    // Build the message NOW, so text and values are from the moment of
    // the fault. PRG_Spray.sErrorText is current: MAIN calls PRG_Spray
    // before this program in the same scan.
    sText := 'SPRAY FAULT ';
    sText := CONCAT(sText, INT_TO_STRING(MAIN.nErrorCode));
    sText := CONCAT(sText, ': ');
    sText := CONCAT(sText, PRG_Spray.sErrorText);
    sText := CONCAT(sText, '\nLevel ');           // '\n' = literal chars
    sText := CONCAT(sText, LREAL_TO_FMTSTR(REAL_TO_LREAL(GVL_IO.rSPXLevel), 1, TRUE));
    sText := CONCAT(sText, ' % / SPX ');
    sText := CONCAT(sText, LREAL_TO_FMTSTR(REAL_TO_LREAL(GVL_IO.rSPXPressure), 2, TRUE));
    sText := CONCAT(sText, ' bar');
    IF fbTime.bValid THEN
        sText := CONCAT(sText, '\n');
        sText := CONCAT(sText, SYSTEMTIME_TO_STRING(fbTime.systemTime));
    END_IF

    // JSON wrapper. The '\n' above is backslash+n (two characters) -
    // JSON turns that into a real newline in the Telegram message.
    // Keep sText plain ASCII without quotes/backslashes, or escape them.
    sPending := '{"chat_id":"';
    sPending := CONCAT(sPending, sChatId);
    sPending := CONCAT(sPending, '","text":"');
    sPending := CONCAT(sPending, sText);
    sPending := CONCAT(sPending, '"}');
    // NOTE: a newer fault overwrites an unsent one (one-slot queue).
END_IF

//==================================================================
// Send state machine: hand over -> wait for the response -> idle.
//==================================================================
CASE eStep OF

    IDLE:
        IF sPending <> '' THEN
            sBody    := sPending;
            sPending := '';
            eStep    := SEND;
        END_IF

    SEND:
        // Retry the handover for up to 10 s (client may still be
        // configuring right after boot), then drop the message.
        tonSendTo(IN := TRUE, PT := T#10S);
        fbRequest.sContentType := 'application/json';
        IF fbRequest.SendRequest(sUri         := sUri,
                                 fbClient     := fbClient,
                                 eRequestType := ETcIotHttpRequestType.HTTP_POST,
                                 pContent     := ADR(sBody),
                                 nContentSize := TO_UDINT(LEN(sBody)),
                                 fbHeader     := 0) THEN
            tonSendTo(IN := FALSE);
            eStep := WAIT_RESPONSE;
        ELSIF tonSendTo.Q THEN
            tonSendTo(IN := FALSE);
            nFailCount := nFailCount + 1;     // never block the machine
            eStep := IDLE;
        END_IF

    WAIT_RESPONSE:
        // bBusy TRUE->FALSE = response received (or the request failed).
        IF NOT fbRequest.bBusy THEN
            nLastStatus := fbRequest.nStatusCode;
            IF fbRequest.bError OR (fbRequest.nStatusCode <> 200) THEN
                nFailCount := nFailCount + 1;
            END_IF
            eStep := IDLE;
        END_IF

END_CASE

END_PROGRAM

// ---- POUs/PRG_StatsLogger.TcPOU
PROGRAM PRG_StatsLogger
VAR
    fbTime     : FB_LocalSystemTime := (bEnable := TRUE, dwCycle := 1);
    tsNow         : TIMESTRUCT;

    // ---- sampling ----
    tonSample  : TON;
    bDue       : BOOL;
    bActive    : BOOL;
    bInWindow  : BOOL;
    tPeriod    : TIME;
    ePrevState : E_SeqState := E_SeqState.eIdle;
    bPrevAuto  : BOOL;

    // ---- time-in-state accumulators (for uptime %) ----
    tonSec     : TON;
    nRunSec    : UDINT;   // resets on PLC restart (by design)
    nIdleSec   : UDINT;
    nFaultSec  : UDINT;

    // ---- line queue (writer drains it; survives short disk hiccups) ----
    aQ         : ARRAY [0..15] OF STRING(255);
    nHead      : INT;
    nTail      : INT;
    nCount     : INT;
    nDropped   : UDINT;

    // ---- file writer state machine ----
    eWr        : (WR_IDLE, WR_OPEN, WR_WRITE, WR_CLOSE);
    fbOpen     : FB_FileOpen;
    fbWrite    : FB_FilePuts;
    fbClose    : FB_FileClose;
    hFile      : UINT;
    bBoot      : BOOL;             // TRUE -> sLogDir='' -> boot folder
    sPath      : STRING(255);
    sLastDate  : STRING(15);
    tonRetry   : TON;
    bBackoff   : BOOL;
    nFailCount : UDINT;
    nLastErrId : UDINT;
    sLastPath  : STRING(255);

    // ---- scratch ----
    sTs        : STRING(63);
    sDate      : STRING(15);
    sFile      : STRING(80);
    sLine      : STRING(255);
    sTail      : STRING(2);
END_VAR

fbTime();

//------------------------------------------------------------------
// 1) time-in-state accumulators (1 s resolution)
//------------------------------------------------------------------
tonSec(IN := NOT tonSec.Q, PT := T#1S);
IF tonSec.Q THEN
    IF MAIN.eState = E_SeqState.eFault THEN
        nFaultSec := nFaultSec + 1;
    ELSIF MAIN.eState = E_SeqState.eIdle THEN
        nIdleSec := nIdleSec + 1;
    ELSE
        nRunSec := nRunSec + 1;
    END_IF
END_IF

//------------------------------------------------------------------
// 2) is logging allowed right now?  (master switch + daily window)
//------------------------------------------------------------------
tsNow := fbTime.systemTime;
IF (GVL_Param.nStatsHourFrom = 0) AND (GVL_Param.nStatsHourTo = 0) THEN
    bInWindow := TRUE;                                   // 24 h logging
ELSIF GVL_Param.nStatsHourFrom <= GVL_Param.nStatsHourTo THEN
    bInWindow := (tsNow.wHour >= INT_TO_WORD(GVL_Param.nStatsHourFrom))
             AND (tsNow.wHour <  INT_TO_WORD(GVL_Param.nStatsHourTo));
ELSE                                                     // window over midnight
    bInWindow := (tsNow.wHour >= INT_TO_WORD(GVL_Param.nStatsHourFrom))
              OR (tsNow.wHour <  INT_TO_WORD(GVL_Param.nStatsHourTo));
END_IF

//------------------------------------------------------------------
// 3) adaptive sample trigger (+ immediate sample on any edge)
//------------------------------------------------------------------
bActive := (MAIN.eState <> E_SeqState.eIdle) AND (MAIN.eState <> E_SeqState.eFault);
tPeriod := SEL(bActive, GVL_Param.tStatsIdle, GVL_Param.tStatsRun);
tonSample(IN := NOT tonSample.Q, PT := tPeriod);
bDue := tonSample.Q;
IF (MAIN.eState <> ePrevState) OR (MAIN.bAutoMode <> bPrevAuto) THEN
    bDue := TRUE;                    // sharp edges on the state timeline
END_IF
ePrevState := MAIN.eState;
bPrevAuto  := MAIN.bAutoMode;

//------------------------------------------------------------------
// 4) build + queue one CSV line
//------------------------------------------------------------------
IF bDue AND bInWindow AND GVL_Param.bStatsEnable AND fbTime.bValid THEN

    // ---- timestamp 'YYYY-MM-DD HH:MM:SS.mmm' (fixed format for Alloy) ----
    sTs := TO_STRING(tsNow.wYear);
    sTs := CONCAT(sTs, SEL(tsNow.wMonth  < 10, '-', '-0'));
    sTs := CONCAT(sTs, TO_STRING(tsNow.wMonth));
    sTs := CONCAT(sTs, SEL(tsNow.wDay    < 10, '-', '-0'));
    sTs := CONCAT(sTs, TO_STRING(tsNow.wDay));
    sDate := sTs;                                        // YYYY-MM-DD
    sTs := CONCAT(sTs, SEL(tsNow.wHour   < 10, ' ', ' 0'));
    sTs := CONCAT(sTs, TO_STRING(tsNow.wHour));
    sTs := CONCAT(sTs, SEL(tsNow.wMinute < 10, ':', ':0'));
    sTs := CONCAT(sTs, TO_STRING(tsNow.wMinute));
    sTs := CONCAT(sTs, SEL(tsNow.wSecond < 10, ':', ':0'));
    sTs := CONCAT(sTs, TO_STRING(tsNow.wSecond));
    sTs := CONCAT(sTs, '.');
    IF tsNow.wMilliseconds < 10 THEN
        sTs := CONCAT(sTs, '00');
    ELSIF tsNow.wMilliseconds < 100 THEN
        sTs := CONCAT(sTs, '0');
    END_IF
    sTs := CONCAT(sTs, TO_STRING(tsNow.wMilliseconds));

    // ---- day rollover: new file name + one header line ----
    IF sDate <> sLastDate THEN
        sLastDate := sDate;
        sFile := CONCAT('machine_stats_', sDate);
        sFile := CONCAT(sFile, '.csv');
        IF GVL_Param.sLogDir = '' THEN
            bBoot := TRUE;
            sPath := sFile;                              // TwinCAT boot folder
        ELSE
            bBoot := FALSE;
            sPath := GVL_Param.sLogDir;
            sTail := RIGHT(sPath, 1);
            IF (sTail <> '\') AND (sTail <> '/') THEN
                sPath := CONCAT(sPath, '/');             // '/' works on Windows too
            END_IF
            sPath := CONCAT(sPath, sFile);
        END_IF
        IF nCount < 16 THEN                              // header line
            aQ[nTail] := '# ts,state,state_n,mode,level_pct,spx_bar,air_bar,pump_hz,err,run_s,idle_s,fault_s';
            nTail := (nTail + 1) MOD 16;
            nCount := nCount + 1;
        END_IF
    END_IF

    // ---- the sample itself ----
    sLine := sTs;
    sLine := CONCAT(sLine, ',');
    sLine := CONCAT(sLine, TO_STRING(MAIN.eState));      // 'eIdle' etc.
    sLine := CONCAT(sLine, ',');
    sLine := CONCAT(sLine, INT_TO_STRING(TO_INT(MAIN.eState)));  // 0/10/../100
    sLine := CONCAT(sLine, SEL(MAIN.bAutoMode, ',MAN', ',AUTO'));
    sLine := CONCAT(sLine, ',');
    sLine := CONCAT(sLine, LREAL_TO_FMTSTR(REAL_TO_LREAL(GVL_IO.rSPXLevel), 1, TRUE));
    sLine := CONCAT(sLine, ',');
    sLine := CONCAT(sLine, LREAL_TO_FMTSTR(REAL_TO_LREAL(GVL_IO.rSPXPressure), 2, TRUE));
    sLine := CONCAT(sLine, ',');
    sLine := CONCAT(sLine, LREAL_TO_FMTSTR(REAL_TO_LREAL(GVL_IO.rAirPressure), 2, TRUE));
    sLine := CONCAT(sLine, ',');
    sLine := CONCAT(sLine, LREAL_TO_FMTSTR(REAL_TO_LREAL(GVL_IO.rPumpHz), 1, TRUE));
    sLine := CONCAT(sLine, ',');
    sLine := CONCAT(sLine, INT_TO_STRING(MAIN.nErrorCode));
    sLine := CONCAT(sLine, ',');
    sLine := CONCAT(sLine, UDINT_TO_STRING(nRunSec));
    sLine := CONCAT(sLine, ',');
    sLine := CONCAT(sLine, UDINT_TO_STRING(nIdleSec));
    sLine := CONCAT(sLine, ',');
    sLine := CONCAT(sLine, UDINT_TO_STRING(nFaultSec));

    IF nCount < 16 THEN
        aQ[nTail] := sLine;
        nTail := (nTail + 1) MOD 16;
        nCount := nCount + 1;
    ELSE
        nDropped := nDropped + 1;                        // disk too slow / stuck
    END_IF
END_IF

//------------------------------------------------------------------
// 5) non-blocking file writer (open -> write all queued -> close)
//------------------------------------------------------------------
CASE eWr OF
    WR_IDLE:
        tonRetry(IN := bBackoff, PT := T#5S);
        IF tonRetry.Q THEN
            bBackoff := FALSE;
        END_IF
        IF (nCount > 0) AND NOT bBackoff AND (sPath <> '') THEN
            sLastPath := sPath;
            eWr := WR_OPEN;
        END_IF

    WR_OPEN:
        fbOpen(sNetId   := '',
               sPathName := sPath,
               nMode    := FOPEN_MODEAPPEND OR FOPEN_MODETEXT,
               ePath    := SEL(bBoot, PATH_GENERIC, PATH_BOOTPATH),
               tTimeout := T#3S,
               bExecute := TRUE);
        IF NOT fbOpen.bBusy THEN
            fbOpen(bExecute := FALSE);
            IF fbOpen.bError THEN
                nLastErrId := fbOpen.nErrId;
                nFailCount := nFailCount + 1;
                bBackoff   := TRUE;
                eWr := WR_IDLE;
            ELSE
                hFile := fbOpen.hFile;
                eWr := WR_WRITE;
            END_IF
        END_IF

    WR_WRITE:
        fbWrite(sNetId   := '',
                hFile    := hFile,
                sLine    := CONCAT(aQ[nHead], '$N'),
                tTimeout := T#3S,
                bExecute := TRUE);
        IF NOT fbWrite.bBusy THEN
            fbWrite(bExecute := FALSE);
            IF fbWrite.bError THEN
                nLastErrId := fbWrite.nErrId;
                nFailCount := nFailCount + 1;
                bBackoff   := TRUE;
                eWr := WR_CLOSE;
            ELSE
                nHead  := (nHead + 1) MOD 16;
                nCount := nCount - 1;
                IF nCount = 0 THEN
                    eWr := WR_CLOSE;
                END_IF
                // else: stay here, next call re-triggers for the next line
            END_IF
        END_IF

    WR_CLOSE:
        fbClose(sNetId   := '',
                hFile    := hFile,
                tTimeout := T#3S,
                bExecute := TRUE);
        IF NOT fbClose.bBusy THEN
            fbClose(bExecute := FALSE);
            IF fbClose.bError THEN
                nLastErrId := fbClose.nErrId;
                nFailCount := nFailCount + 1;
            END_IF
            hFile := 0;
            eWr := WR_IDLE;
        END_IF
END_CASE

END_PROGRAM

// ---- GlobalTextList.TcGTLO
TEXTLIST GlobalTextList
  14 = '%.0f'
  367 = '%.0f Hz'
  546 = '%.1f'
  942 = '%s'
  399 = 'Add Water'
  603 = 'air valve'
  116 = 'Air: %.2f bar'
  911 = 'apply'
  134 = 'Bar'
  53 = 'Circulation'
  917 = 'Circulation and feeding'
  709 = 'clean mode'
  117 = 'close'
  141 = 'Close Drain'
  898 = 'Error: %s'
  302 = 'Home page'
  563 = 'Hz'
  863 = 'j'
  802 = 'Label'
  962 = 'Machine Parameters'
  80 = 'Manual / Auto'
  899 = 'Manual page'
  926 = 'open'
  531 = 'Open Air Valve'
  412 = 'Open SPX Valve'
  656 = 'Parameters'
  730 = 'Piston '
  619 = 'PRG_Spray.sModeText'
  122 = 'pump'
  499 = 'Pump speed'
  931 = 'pump speed'
  295 = 'Reset'
  775 = 'RESET DEFAULTS'
  560 = 'Run Pump'
  450 = 's'
  919 = 'S'
  518 = 'sim/real value'
  989 = 'Spray System'
  187 = 'spx level'
  132 = 'SPX Pressure target'
  488 = 'SPX valve'
  925 = 'SPX: %.2f bar'
  495 = 'Start Clean'
  998 = 'State: %s'
  15 = 'StepNo: %d'
  394 = 'Switch to Manual mode to edit parameters'
  535 = 'T1 : Dewater time'
  84 = 'T2 & T6 : Valve max open/close'
  304 = 'T3 & T4 : Max spraying time'
  12 = 'T5 : SPX Dewater time'
END_TEXTLIST

// ---- VISUs/visu_Nav.TcVIS
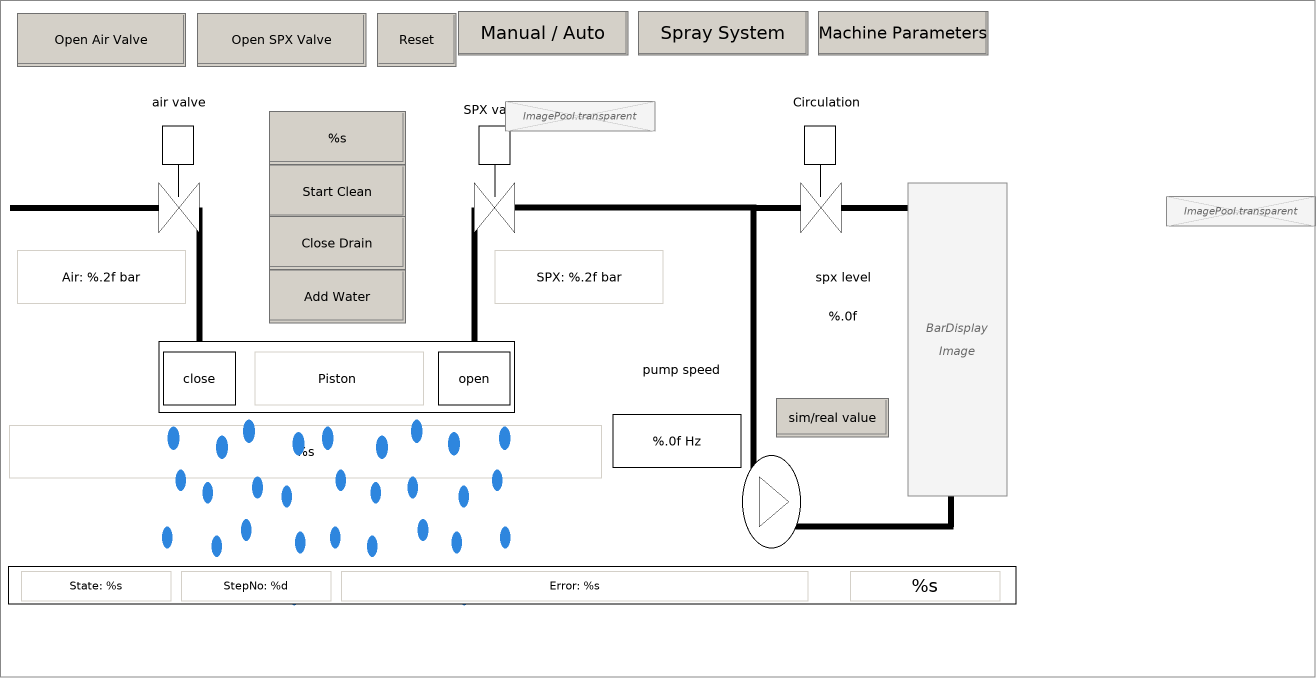
VISUALIZATION visu_Nav  // 1316x678
AR_IN_OUT
	
END_VAR
    Frame (8,-1 999x549), frame switch variable: GVL_Nav.nPage
        shows visu_Spray()
        shows visu_Params()
    Button (638,11 170x44), "Spray System"
        p2175578022: SEL(GVL_Nav.abNavActive[0], 16#FF2D6FE0, 16#FF1FA34A)
        OnMouseClick: FrameSelectionChange Selection=SelectedFrame=ec7dd251-7f6b-4bd4-83c6-e8d232fe81a4, GlobSel=IndExpr=0, AssignType=Expression, SelType=Globally, SelectionStep=SelectedAction=SwitchNext
        OnMouseClick: execute { GVL_Nav.nPage := 0; }
    Button (818,11 170x44), "Machine Parameters"
        p2175578022: SEL(GVL_Nav.abNavActive[1], 16#FF2D6FE0, 16#FF1FA34A)
        OnMouseClick: FrameSelectionChange Selection=Selection=-1, GlobSel=IndExpr=1, AssignType=Expression, SelType=Globally, SelectionStep=SelectedAction=SwitchNext
        OnMouseClick: execute { GVL_Nav.nPage := 1; }
    Rectangle (8,566 1008x38)
    Textfield (21,571 150x30), "State: %s", text variable: PRG_Spray.sStateText
    Textfield (181,571 150x30), "StepNo: %d", text variable: TO_INT(MAIN.eState)
    Textfield (341,571 467x30), "Error: %s", text variable: PRG_Spray.sErrorText
    Textfield (850,571 150x30), "%s", text variable: PRG_Spray.sModeText
        p55702900: PRG_Spray.cModeColor
    Button (458,11 170x44), "Manual / Auto"
        p2175578022: PRG_Spray.cModeColor
        OnMouseClick: toggle PRG_Spray.bCmdAuto
    Line (956,676)
    Image (505,101 150x30), image: ImagePool.transparent
    Image (1166,196 150x30), image: ImagePool.transparent
END_VISUALIZATION

// ---- VISUs/visu_Params.TcVIS
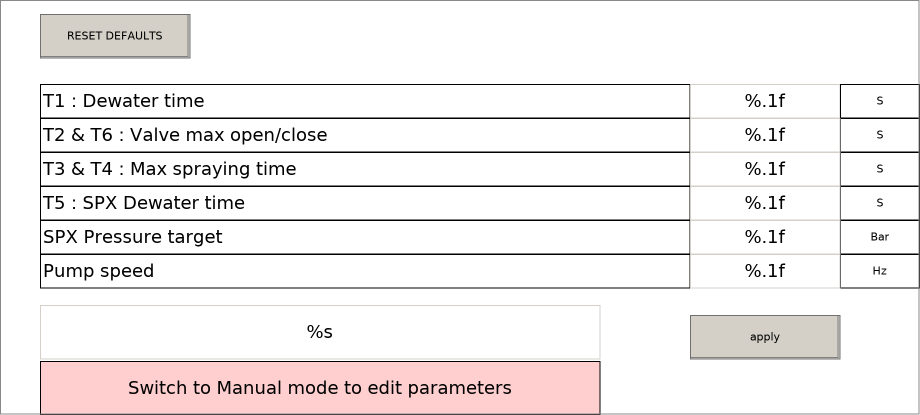
VISUALIZATION visu_Params  // 920x415
    Rectangle (40,84 650x34), "T1 : Dewater time"
    Textfield (690,84 150x34), "%.1f", text variable: PRG_Params.rEditDewater_s, input disabled if: NOT PRG_Spray.bManualActive
        OnMouseClick: write the text variable via VisuDialogs.Numpad, min 0, max 9999999
    Rectangle (840,84 80x34), "S"
    Rectangle (840,118 80x34), "S"
    Rectangle (40,118 650x34), "T2 & T6 : Valve max open/close"
    Textfield (690,118 150x34), "%.1f", text variable: PRG_Params.rEditValveMax_s, input disabled if: NOT PRG_Spray.bManualActive
        OnMouseClick: write the text variable via VisuDialogs.Numpad, min 0, max 9999999
    Rectangle (840,152 80x34), "S"
    Rectangle (40,152 650x34), "T3 & T4 : Max spraying time"
    Textfield (690,152 150x34), "%.1f", text variable: PRG_Params.rEditSprayTime_s, input disabled if: NOT PRG_Spray.bManualActive
        OnMouseClick: write the text variable via VisuDialogs.Numpad, min 0, max 9999999
    Rectangle (840,186 80x34), "S"
    Rectangle (40,186 650x34), "T5 : SPX Dewater time"
    Textfield (690,186 150x34), "%.1f", text variable: PRG_Params.rEditSPXDewater_s, input disabled if: NOT PRG_Spray.bManualActive
        OnMouseClick: write the text variable via VisuDialogs.Numpad, min 0, max 9999999
    Rectangle (840,220 80x34), "Bar"
    Rectangle (40,220 650x34), "SPX Pressure target"
    Textfield (690,220 150x34), "%.1f", text variable: PRG_Params.rEditPressTarget, input disabled if: NOT PRG_Spray.bManualActive
        OnMouseClick: write the text variable via VisuDialogs.Numpad, min 0, max 9999999
    Rectangle (840,254 80x34), "Hz"
    Rectangle (40,254 650x34), "Pump speed"
    Textfield (690,254 150x34), "%.1f", text variable: PRG_Params.rEditPumpSpeed, input disabled if: NOT PRG_Spray.bManualActive
        OnMouseClick: write the text variable via VisuDialogs.Numpad, min 0, max 9999999
    Button (690,315 150x44), "apply", input disabled if: NOT PRG_Spray.bManualActive
        tap PRG_Params.bBtnApply
    Textfield (40,305 560x54), "%s", text variable: PRG_Params.sParamStatus, invisible if: NOT PRG_Params.bMsgVisible
    Rectangle (40,361 560x54), "Switch to Manual mode to edit parameters", invisible if: NOT (PRG_Params.bMsgVisible AND NOT PRG_Spray.bManualActive)
    Button (40,14 150x44), "RESET DEFAULTS", input disabled if: NOT PRG_Spray.bManualActive
        tap PRG_Params.bBtnReset
END_VISUALIZATION

// ---- VISUs/visu_Spray.TcVIS
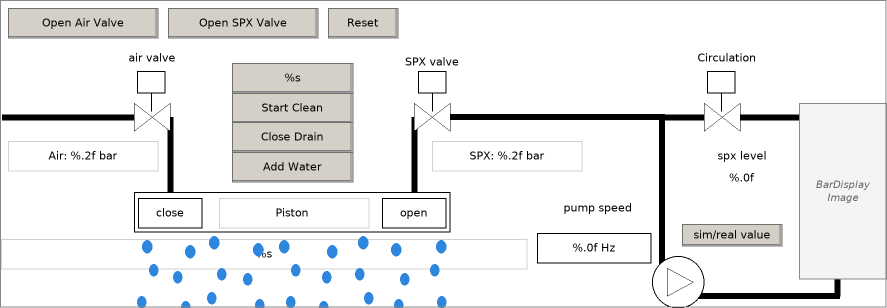
VISUALIZATION visu_Spray  // 887x308
    Button (8,8 150x30), "Open Air Valve", input disabled if: NOT PRG_Spray.bManualActive
        toggle PRG_Spray.bManAirValve p2164770859=TRUE
    Button (168,8 150x30), "Open SPX Valve", input disabled if: NOT PRG_Spray.bManualActive
        toggle PRG_Spray.bManSPXValve
    Button (328,8 70x30), "Reset"
        tap PRG_Spray.bCmdReset
    Polyline (2,117) (134,117)
    Polyline (170,117) (170,200)
    Polyline (414,117) (414,200)
    Polyline (662,117) (704,117)
    Polyline (662,269) (662,117) (450,117)
    Polyline (740,117) (837,117) (837,117)
    Polyline (837,265) (837,296) (690,296)
    Polygon (414,103) (450,131) (450,103) (414,131), colour variable: PRG_Spray.cSPXValve
    Polygon (704,103) (740,131) (740,103) (704,131), colour variable: PRG_Spray.cCircValve
    Line (432,93) (432,111)
    Rectangle (418,71 28x22), colour variable: PRG_Spray.cSPXValve
    Label (102,49 100x18), "air valve"
    Label (357,53 150x18), "SPX valve"
    Label (677,49 100x18), "Circulation"
    Rectangle (537,233 114x30), "%.0f Hz", text variable: GVL_IO.rPumpHz
    RoundedRectangle (134,192 316x40)
    Textfield (219,198 150x30), "Piston"
    Rectangle (138,198 64x30), "close", colour variable: PRG_Spray.cPistonClose
    Rectangle (382,198 64x30), "open", colour variable: PRG_Spray.cPistonOpen
    Ellipse (652,256 52x52)
    Polygon (667,268) (667,296) (693,282)
    Label (523,193 150x30), "pump speed"
    Textfield (704,163 75x30), "%.0f", text variable: GVL_IO.rSPXLevel
        p55702900: PRG_Spray.cLevel
    Line (721,93) (721,111)
    Rectangle (707,71 28x22), colour variable: PRG_Spray.cCircValve
    Line (151,93) (151,111)
    Rectangle (137,71 28x22), colour variable: PRG_Spray.cAirValve
    Polygon (134,103) (170,131) (170,103) (134,131), colour variable: PRG_Spray.cAirValve
    Label (667,141 150x30), "spx level"
    Button (682,224 100x22), "sim/real value"
        OnMouseClick: toggle SIM_Plant.bSimLevelActive
    BarDisplayImage (799,103 88x176), value: GVL_IO.rSPXLevel, style: BarDisplayImage-Green, scale format: %.0f, scale 0..100
    Button (232,63 121x30), "%s", text variable: PRG_Spray.sCleanBtnText, invisible if: NOT PRG_Spray.bManualActive
        toggle PRG_Spray.bBtnClean
    Button (232,93 121x30), "Start Clean", invisible if: NOT PRG_Spray.bCleanActive
        toggle PRG_Spray.bBtnStartClean
    Button (232,122 121x30), "Close Drain", colour toggle: PRG_Spray.bDrainFlash, invisible if: NOT PRG_Spray.bCleanActive
        toggle PRG_Spray.bBtnCloseDrain
    Button (232,152 121x30), "Add Water", colour toggle: PRG_Spray.bWaterFlash, invisible if: NOT PRG_Spray.bCleanActive
        toggle PRG_Spray.bBtnAddWater
    Textfield (1,239 526x30), "%s", text variable: PRG_Spray.sCleanStatus, invisible if: NOT PRG_Spray.bCleanActive
    Textfield (432,141 150x30), "SPX: %.2f bar", text variable: GVL_IO.rSPXPressure
        p55702900: PRG_Spray.cSPXPress
    Textfield (8,141 150x30), "Air: %.2f bar", text variable: GVL_IO.rAirPressure
    Ellipse (142,240 10x13), invisible if: NOT PRG_Spray.abDrop[0]
    Ellipse (185,245 10x13), invisible if: NOT PRG_Spray.abDrop[1]
    Ellipse (209,236 10x13), invisible if: NOT PRG_Spray.abDrop[2]
    Ellipse (253,243 10x13), invisible if: NOT PRG_Spray.abDrop[3]
    Ellipse (279,240 10x13), invisible if: NOT PRG_Spray.abDrop[0]
    Ellipse (327,245 10x13), invisible if: NOT PRG_Spray.abDrop[1]
    Ellipse (358,236 10x13), invisible if: NOT PRG_Spray.abDrop[2]
    Ellipse (391,243 10x13), invisible if: NOT PRG_Spray.abDrop[3]
    Ellipse (436,240 10x13), invisible if: NOT PRG_Spray.abDrop[0]
    Ellipse (149,264 9x12), invisible if: NOT PRG_Spray.abDrop[1]
    Ellipse (173,271 9x12), invisible if: NOT PRG_Spray.abDrop[2]
    Ellipse (217,268 9x12), invisible if: NOT PRG_Spray.abDrop[3]
    Ellipse (243,273 9x12), invisible if: NOT PRG_Spray.abDrop[0]
    Ellipse (291,264 9x12), invisible if: NOT PRG_Spray.abDrop[1]
    Ellipse (322,271 9x12), invisible if: NOT PRG_Spray.abDrop[2]
    Ellipse (355,268 9x12), invisible if: NOT PRG_Spray.abDrop[3]
    Ellipse (400,273 9x12), invisible if: NOT PRG_Spray.abDrop[0]
    Ellipse (430,264 9x12), invisible if: NOT PRG_Spray.abDrop[1]
    Ellipse (137,296 9x12), invisible if: NOT PRG_Spray.abDrop[2]
    Ellipse (181,301 9x12), invisible if: NOT PRG_Spray.abDrop[3]
    Ellipse (207,292 9x12), invisible if: NOT PRG_Spray.abDrop[0]
    Ellipse (255,299 9x12), invisible if: NOT PRG_Spray.abDrop[1]
    Ellipse (286,296 9x12), invisible if: NOT PRG_Spray.abDrop[2]
    Ellipse (319,301 9x12), invisible if: NOT PRG_Spray.abDrop[3]
    Ellipse (364,292 9x12), invisible if: NOT PRG_Spray.abDrop[0]
    Ellipse (394,299 9x12), invisible if: NOT PRG_Spray.abDrop[1]
    Ellipse (437,296 9x12), invisible if: NOT PRG_Spray.abDrop[2]
    Ellipse (145,320 8x11), invisible if: NOT PRG_Spray.abDrop[3]
    Ellipse (171,327 8x11), invisible if: NOT PRG_Spray.abDrop[0]
    Ellipse (219,324 8x11), invisible if: NOT PRG_Spray.abDrop[1]
    Ellipse (250,329 8x11), invisible if: NOT PRG_Spray.abDrop[2]
    Ellipse (283,320 8x11), invisible if: NOT PRG_Spray.abDrop[3]
    Ellipse (328,327 8x11), invisible if: NOT PRG_Spray.abDrop[0]
    Ellipse (358,324 8x11), invisible if: NOT PRG_Spray.abDrop[1]
    Ellipse (401,329 8x11), invisible if: NOT PRG_Spray.abDrop[2]
    Ellipse (425,320 8x11), invisible if: NOT PRG_Spray.abDrop[3]
END_VISUALIZATION
